// TwinCAT 3 PLC project plc_dream_gsjn_test
// ProgramVersion: 3.1.4022.7
// libraries:
//   LCLS General, * (SLAC)
//   lcls-twincat-motion, * (SLAC)
//   PMPS, * (SLAC - LCLS)
//   Tc2_Standard, * (Beckhoff Automation GmbH)
//   Tc2_System, * (Beckhoff Automation GmbH)
//   Tc3_Module, * (Beckhoff Automation GmbH)
// project tree:
//   GVLs/ GVL_Devices.TcGVL
//   / PlcTask.TcTTO
//   POUs/ MAIN.TcPOU
// real-time tasks:
//   TASK PlcTask: cycle T#10ms, priority 20, ADS port 350
// motion (NC):
// I/O:
//   DEVICE Device 1 (EtherCAT), AmsNetId 172.21.132.189.2.1
//     Term 1 (EK1200) [EK1200-5000 EtherCAT Power supply (2A E-Bus)]
//       Term 2 (EL7047)
//       Term 3 (EL5042) [EL5042 2Ch. BiSS-C Encoder]
//       Term 4 (EL2004) [EL2004 4Ch. Dig. Output 24V, 0.5A]
//       Term 5 (EL3064) [EL3064 4Ch. Ana. Input 0-10V]
//       Term 6 (EK1110)
// variable links:
//   plc_dream_gsjn_test Instance <-> Device 1 (EtherCAT)/Term 1 (EK1200)/Term 2 (EL7047)
//     PlcTask Inputs/GVL_Devices.M1.bLimitBackwardEnable <-> STM Status/Status/Digital input 2
//     PlcTask Inputs/GVL_Devices.M1.bLimitForwardEnable <-> STM Status/Status/Digital input 1
//   plc_dream_gsjn_test Instance <-> Device 1 (EtherCAT)/Term 1 (EK1200)/Term 3 (EL5042)
//     PlcTask Inputs/GVL_Devices.M1.nRawEncoderULINT <-> FB Inputs Channel 2/Position

CONFIGURATION plc_dream_gsjn_test
    RESOURCE PLC ON TwinCAT3
        TASK PlcTask(INTERVAL := T#10ms, PRIORITY := 20);
        PROGRAM MAIN WITH PlcTask : MAIN;
    END_RESOURCE
END_CONFIGURATION

// ---- GVLs/GVL_Devices.TcGVL
VAR_GLOBAL
    bLimitForward AT %Q* : BOOL := TRUE;
    bLimitBackward AT %Q* : BOOL := TRUE;

    eStageEnableMode : ENUM_StageEnableMode := ENUM_StageEnableMode.DURING_MOTION;
    {attribute 'TcLinkTo' := '.bLimitForwardEnable  := TIIB[Term 2 (EL7047)]^STM Status^Status^Digital input 1;
                              .bLimitBackwardEnable := TIIB[Term 2 (EL7047)]^STM Status^Status^Digital input 2;
                              .nRawEncoderULINT     := TIIB[Term 3 (EL5042)]^FB Inputs Channel 2^Position'}
    {attribute 'pytmc' := '
        pv: TST:LAB:MMS:01
    '}
    M1: ST_MotionStage := (
        bHardwareEnable := TRUE,
        bPowerSelf := TRUE,
        nEnableMode := eStageEnableMode,
        nHomingMode := ENUM_EpicsHomeCmd.NONE,
        sName := 'TST:LAB:MMS:01');
END_VAR

// ---- POUs/MAIN.TcPOU
PROGRAM MAIN
VAR
    fbMotionTstLab: FB_MotionStage;
END_VAR

//Run fb Motion Stage
fbMotionTstLab(stMotionStage:=GVL_Devices.M1);

END_PROGRAM
